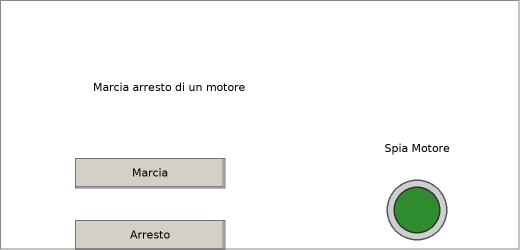
VISUALIZATION Visualization  // 520x250
    Label (67,66 205x43), "Marcia arresto di un motore"
    Button (75,158 150x30), "Marcia", colour toggle: GVL.StartMotor
        tap GVL.StartMotor
    Button (75,220 150x30), "Arresto", colour toggle: GVL.StopMotor
        tap GVL.StopMotor
    Lamp1 (382,175 70x70), variable: GVL.MotorActive, style: Lamp-Lamp1-Green
    Label (315,127 205x43), "Spia Motore"
END_VISUALIZATION

(* stored: Version 1.1.0.1, ProductVersion 3.1.4024.12
   Visu Visualization: Id {2a3825bd-3fd3-4623-9b7a-72538f57fba8} *)
